SUBAPPLICATION mapping_DataPanel_QX (* Subapplication Type *)
  (* Standard: 61499-2 *)
  (* Version 1.0, 2023-01-29, Franz *)
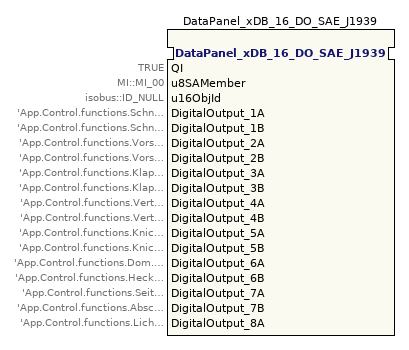
  FBS
    DataPanel_xDB_16_DO_SAE_J1939 : DataPanel_xDB_16_DO_SAE_J1939(QI := TRUE, u8SAMember := MI::MI_00, u16ObjId := isobus::ID_NULL, DigitalOutput_1A := 'App.Control.functions.Schneidwerk.rechtslauf', DigitalOutput_1B := 'App.Control.functions.Schneidwerk.linkslauf', DigitalOutput_2A := 'App.Control.functions.Vorsteuerventil_2A.QX', DigitalOutput_2B := 'App.Control.functions.Vorsteuerventil_2B.QX', DigitalOutput_3A := 'App.Control.functions.Klappen.Sitzventile.QXA', DigitalOutput_3B := 'App.Control.functions.Klappen.Sitzventile.QXB', DigitalOutput_4A := 'App.Control.functions.Verteiler.Sitzventile.QXA', DigitalOutput_4B := 'App.Control.functions.Verteiler.Sitzventile.QXB', DigitalOutput_5A := 'App.Control.functions.Knickdeichsel.Sitzventile.QXA', DigitalOutput_5B := 'App.Control.functions.Knickdeichsel.Sitzventile.QXB', DigitalOutput_6A := 'App.Control.functions.Dom.QX', DigitalOutput_6B := 'App.Control.functions.Heckschieber.QXB', DigitalOutput_7A := 'App.Control.functions.Seitenschieber.QX', DigitalOutput_7B := 'App.Control.functions.Abscheider.QX', DigitalOutput_8A := 'App.Control.functions.Licht.QX');
  END_FBS
END_SUBAPPLICATION
